# EPICS substitutions: db/Beckhoff_1XXX/ecmcEL1862.substitutions
# generic slave part
file "ecmcEcSlave.template"{
  pattern {}
          {}
}

# binary inputs
file "ecmc_binaryInput-chX.template"{
  pattern {CH_ID}
          {01   }
          {02   }
          {03   }
          {04   }
          {05   }
          {06   }
          {07   }
          {08   }
          {09   }
          {10   }
          {11   }
          {12   }
          {13   }
          {14   }
          {15   }
          {16   }
}
